{attribute addProperty BoxType "EL1512-0000-0017"}
{attribute addProperty Id "Set_counter_doneBIT10.1253Counter_inhibitedBIT10.1254Status_of_input_clockBIT10.1256TxPDO_ToggleBIT10.1259"}
{attribute addProperty CRC "3648402039"}
{attribute addProperty SizeInBites "16"}
{attribute addProperty SizeInBytes "2"}
TYPE Status_D9763277 :
STRUCT
	{attribute 'hide'}
	reserve_1_BIT_0 : BIT;
	{attribute 'hide'}
	reserve_1_BIT_1 : BIT;
	{attribute addProperty Name "Set_counter_done"}
	Set_counter_done : BIT;
	{attribute addProperty Name "Counter_inhibited"}
	Counter_inhibited : BIT;
	{attribute 'hide'}
	reserve_2 : BIT;
	{attribute addProperty Name "Status_of_input_clock"}
	Status_of_input_clock : BIT;
	{attribute 'hide'}
	reserve_3_BIT_0 : BIT;
	{attribute 'hide'}
	reserve_3_BIT_1 : BIT;
	{attribute 'hide'}
	reserve_3_BIT_2 : BIT;
	{attribute 'hide'}
	reserve_3_BIT_3 : BIT;
	{attribute 'hide'}
	reserve_3_BIT_4 : BIT;
	{attribute 'hide'}
	reserve_3_BIT_5 : BIT;
	{attribute 'hide'}
	reserve_3_BIT_6 : BIT;
	{attribute 'hide'}
	reserve_3_BIT_7 : BIT;
	{attribute 'hide'}
	reserve_3_BIT_8 : BIT;
	{attribute addProperty Name "TxPDO_Toggle"}
	TxPDO_Toggle : BIT;
END_STRUCT
END_TYPE

(* stored: Version 1.2.0.0, ProductVersion 3.1.4024.9
   DUT Status_D9763277: Id {fda3382d-1dfb-4fe6-9bfb-fd1beef25a02} *)
